Staubli VAL3: page.pjx

--- page.pjx ---
Parameters version=s7.2.1 stackSize=50000 millimeterUnit=true
Program file=main.pgx
Data file=page.dtx
Library alias=io path=Disk://io/io.pjx

--- page.dtx ---
public string sItems

--- main.pgx ---
public program main()
  local num lKey
begin
end
